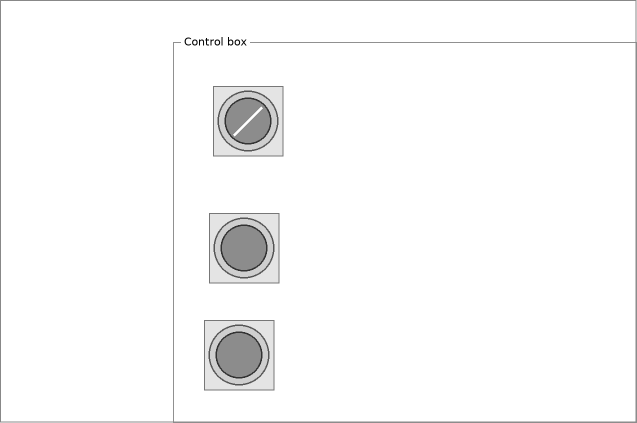
VISUALIZATION Visualization  // 637x423
    GroupBox (173,34 464x389), "Control box"
        PushSwitch (36,179 70x70), behaviour: TOGGLE, style: Switch-PushSwitch-Gray
        PushSwitch (31,286 70x70), variable: GVL.start_Button, behaviour: TOGGLE, style: Switch-PushSwitch-Gray
        RotarySwitch (40,52 70x70), variable: GVL.jijiji, behaviour: TOGGLE, style: Switch-RotarySwitch-Gray
END_VISUALIZATION

(* stored: Version 1.1.0.1, ProductVersion 3.1.4024.12
   Visu Visualization: Id {8cbeb44e-ab14-4ef2-98ed-ba1e56cddae9} *)
